Staubli VAL3: remMovXYZ.pgx

program remMovXYZ(string& sArgs[] (dimensions=1), string& sReturn[] (dimensions=1))
  local bool bOk
  local num nLoop
  local num nVal
  local string sArgsLoop
  local trsf trDest
begin
  // Move to the designated point.
  //
  // Arguments are "X Y Z RX RY RZ"
  //
  logMsg("call remMovXYZ")
  //break down our 6 args and make sure they are numbers
  trDest={0,0,0,0,0,0}
  nLoop=0
  sArgsLoop=sArgs
  while nLoop<6
    sArgsLoop=toNum(sArgsLoop,nVal,bOk)
    if bOk
      switch nLoop
        case 0
          trDest.x=nVal
        break
        case 1
          trDest.y=nVal
        break
        case 2
          trDest.z=nVal
        break
        case 3
          trDest.rx=nVal
        break
        case 4
          trDest.ry=nVal
        break
        case 5
          trDest.rz=nVal
        break
      endSwitch
      nLoop=nLoop+1
    else
      call remErrNum("MOVXYZ",sArgs,sReturn)
      return
    endIf
  endWhile
  call remMovPoint(trDest,sReturn)
end
